# EPICS substitutions: ioc/PSCApp/Db/inp_register.substitutions
file db/inp_register.db {
    pattern {INP_REGISTER_NUMBER}
        {"1"}
}
